{attribute 'hide'}
FUNCTION_BLOCK Test_MultipleNotificationsWithStringArgs EXTENDS T_UnitTestBase
VAR
    Source  : T_Notification;
    Handler : T_NotificationHandler;

    IsRaised          : BOOL;
    NotificationCount : DINT;
	Assertion : T_Assertion;
END_VAR

{attribute 'analysis' := '-33'} // inhibit unused variable warning
METHOD RunTest
VAR_OUTPUT
    TestCompleted : BOOL;
    TestFailed    : BOOL;
END_VAR
Handler.FB_init(bInitRetains := FALSE,
                bInCopyCode  := FALSE);

IsRaised          := FALSE;
NotificationCount := 0;

Source.ClearNotificationHandlers().AddNotificationHandler(Handler);
Source.Args.Init(8);

Source.Args.Clear()
    .Add_INT(1234).Add_STRING('String1');

Source.Raise();

Source.Args.Clear()
    .Add_INT(5678).Add_STRING('String2');

Source.Raise();

TestFailed S= NOT Assertion.AssertEquals_DINT(Source    := TestName,
                             Expected     := 2,
                            Actual       := Handler.NotificationCount,
                            VariableName := 'Handler.NotificationCount');

TestFailed S= NOT Assertion.AssertEquals_BOOL(Source    := TestName,
                             Expected     := TRUE,
                            Actual       := Handler.IsRaised(),
                            VariableName := 'Handler.IsRaised()');

TestFailed S= NOT Assertion.AssertEquals_DINT(Source    := TestName,
                             Expected     := 1,
                            Actual       := Handler.NotificationCount,
                            VariableName := 'Handler.NotificationCount');

TestFailed S= NOT Assertion.AssertEquals_DINT(Source    := TestName,
                             Expected     := 1234,
                            Actual       := Handler.Args.Read_INT(),
                            VariableName := 'Handler.Args.Read_INT()');

TestFailed S= NOT Assertion.AssertEquals_STRING(Source    := TestName,
                             Expected     := 'String1',
                              Actual       := Handler.Args.Read_STRING(),
                              VariableName := 'Handler.Args.Read_STRING()');

TestFailed S= NOT Assertion.AssertEquals_BOOL(Source    := TestName,
                             Expected     := TRUE,
                            Actual       := Handler.IsRaised(),
                            VariableName := 'Handler.IsRaised()');

TestFailed S= NOT Assertion.AssertEquals_DINT(Source    := TestName,
                             Expected     := 0,
                            Actual       := Handler.NotificationCount,
                            VariableName := 'Handler.NotificationCount');

TestFailed S= NOT Assertion.AssertEquals_DINT(Source    := TestName,
                             Expected     := 5678,
                            Actual       := Handler.Args.Read_INT(),
                            VariableName := 'Handler.Args.Read_INT()');

TestFailed S= NOT Assertion.AssertEquals_STRING(Source    := TestName,
                             Expected     := 'String2',
                              Actual       := Handler.Args.Read_STRING(),
                              VariableName := 'Handler.Args.Read_STRING()');

TestFailed S= NOT Assertion.AssertEquals_BOOL(Source    := TestName,
                             Expected     := FALSE,
                            Actual       := Handler.IsRaised(),
                            VariableName := 'Handler.IsRaised()');

TestCompleted := TRUE;
END_METHOD

END_FUNCTION_BLOCK

(* stored: Version 1.1.0.1, ProductVersion 3.1.4024.12
   POU Test_MultipleNotificationsWithStringArgs: Id {498ab529-1915-457a-a89d-d6efea9df911}, SpecialFunc None
   Method RunTest: Id {31f34b70-06bc-4dfb-bb6b-2d182b20f751} *)
